PROGRAM PRG_PLAS_15_PrimaryMasterListCtrl
VAR

	bEnablePackMasterListCameraSystem 	: BOOL;

	tofPrimaryMasterListCameraOFFDelay 		: TOF;

	fbShiftMasterListQueue			: FB_PLAS_MasterListShiftQueue;
	fbPrimaryMasterListCamera		: FB_SCANNER_CameraSelect;
	fbPrimaryMasterListEvaluation		: FB_SCANNER_Evaluation;

	fbAddToPrimaryListQueue			: FB_PLAS_MasterListAddToQueue;

	rtrigNewArrived					: R_TRIG;
	bNewCodeIsProccesing			: BOOL;

	tonValidationTimout				: TON;
	bValidationTimeout				: BOOL;
	bValidationTimeoutReset			: BOOL;

	rtPrimaryMasterListCameraDone		:  R_TRIG;
	bPrimaryMasterListCameraDone		:  BOOL;

	fbDebugCNT						: FB_DEBUG_CounterArray;
	aCNTDebug						: ARRAY [1..10] OF UDINT;
	bResetCNT							: BOOL;

END_VAR

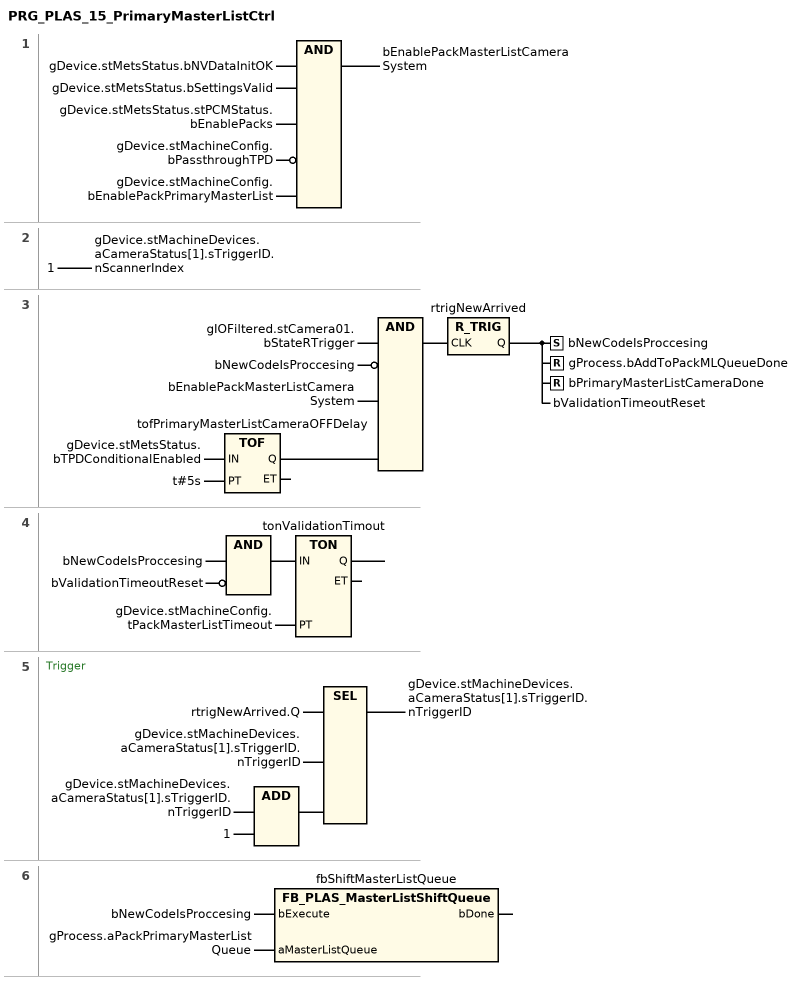
// NETWORK 1
bEnablePackMasterListCameraSystem := gDevice.stMetsStatus.bNVDataInitOK AND gDevice.stMetsStatus.bSettingsValid AND gDevice.stMetsStatus.stPCMStatus.bEnablePacks AND NOT gDevice.stMachineConfig.bPassthroughTPD AND gDevice.stMachineConfig.bEnablePackPrimaryMasterList;

// NETWORK 2
gDevice.stMachineDevices.aCameraStatus[1].sTriggerID.nScannerIndex := 1;

// NETWORK 3
tofPrimaryMasterListCameraOFFDelay(IN := gDevice.stMetsStatus.bTPDConditionalEnabled, PT := t#5s); // TOF
rtrigNewArrived(CLK := gIOFiltered.stCamera01.bStateRTrigger AND NOT bNewCodeIsProccesing AND bEnablePackMasterListCameraSystem AND tofPrimaryMasterListCameraOFFDelay.Q); // R_TRIG
bNewCodeIsProccesing S= rtrigNewArrived.Q;
gProcess.bAddToPackMLQueueDone R= rtrigNewArrived.Q;
bPrimaryMasterListCameraDone R= rtrigNewArrived.Q;
bValidationTimeoutReset := rtrigNewArrived.Q;

// NETWORK 4
tonValidationTimout(IN := bNewCodeIsProccesing AND NOT bValidationTimeoutReset, PT := gDevice.stMachineConfig.tPackMasterListTimeout); // TON

// NETWORK 5
// Trigger
gDevice.stMachineDevices.aCameraStatus[1].sTriggerID.nTriggerID := SEL(rtrigNewArrived.Q, gDevice.stMachineDevices.aCameraStatus[1].sTriggerID.nTriggerID, gDevice.stMachineDevices.aCameraStatus[1].sTriggerID.nTriggerID + 1);

// NETWORK 6
fbShiftMasterListQueue(bExecute := bNewCodeIsProccesing, aMasterListQueue := gProcess.aPackPrimaryMasterListQueue); // FB_PLAS_MasterListShiftQueue

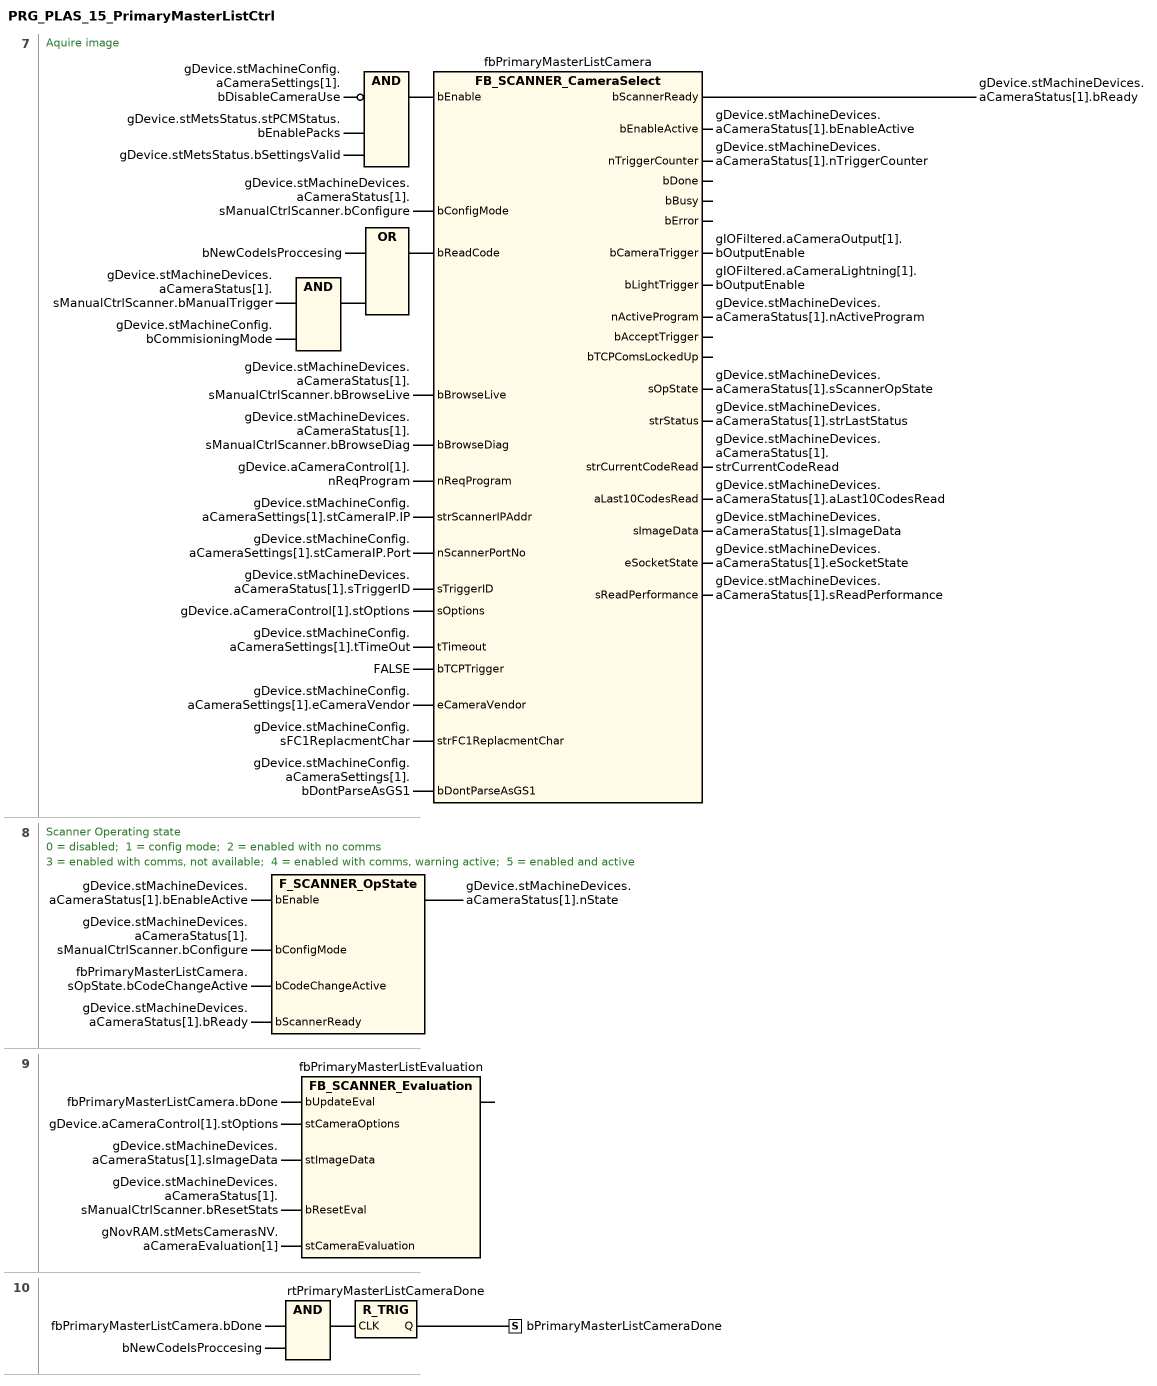
// NETWORK 7
// Aquire image
fbPrimaryMasterListCamera(
    bEnable := NOT gDevice.stMachineConfig.aCameraSettings[1].bDisableCameraUse AND gDevice.stMetsStatus.stPCMStatus.bEnablePacks AND gDevice.stMetsStatus.bSettingsValid,
    bConfigMode := gDevice.stMachineDevices.aCameraStatus[1].sManualCtrlScanner.bConfigure,
    bReadCode := bNewCodeIsProccesing OR gDevice.stMachineDevices.aCameraStatus[1].sManualCtrlScanner.bManualTrigger AND gDevice.stMachineConfig.bCommisioningMode,
    bBrowseLive := gDevice.stMachineDevices.aCameraStatus[1].sManualCtrlScanner.bBrowseLive,
    bBrowseDiag := gDevice.stMachineDevices.aCameraStatus[1].sManualCtrlScanner.bBrowseDiag,
    nReqProgram := gDevice.aCameraControl[1].nReqProgram,
    strScannerIPAddr := gDevice.stMachineConfig.aCameraSettings[1].stCameraIP.IP,
    nScannerPortNo := gDevice.stMachineConfig.aCameraSettings[1].stCameraIP.Port,
    sTriggerID := gDevice.stMachineDevices.aCameraStatus[1].sTriggerID,
    sOptions := gDevice.aCameraControl[1].stOptions,
    tTimeout := gDevice.stMachineConfig.aCameraSettings[1].tTimeOut,
    bTCPTrigger := FALSE,
    eCameraVendor := gDevice.stMachineConfig.aCameraSettings[1].eCameraVendor,
    strFC1ReplacmentChar := gDevice.stMachineConfig.sFC1ReplacmentChar,
    bDontParseAsGS1 := gDevice.stMachineConfig.aCameraSettings[1].bDontParseAsGS1,
    bEnableActive => gDevice.stMachineDevices.aCameraStatus[1].bEnableActive,
    nTriggerCounter => gDevice.stMachineDevices.aCameraStatus[1].nTriggerCounter,
    bCameraTrigger => gIOFiltered.aCameraOutput[1].bOutputEnable,
    bLightTrigger => gIOFiltered.aCameraLightning[1].bOutputEnable,
    nActiveProgram => gDevice.stMachineDevices.aCameraStatus[1].nActiveProgram,
    sOpState => gDevice.stMachineDevices.aCameraStatus[1].sScannerOpState,
    strStatus => gDevice.stMachineDevices.aCameraStatus[1].strLastStatus,
    strCurrentCodeRead => gDevice.stMachineDevices.aCameraStatus[1].strCurrentCodeRead,
    aLast10CodesRead => gDevice.stMachineDevices.aCameraStatus[1].aLast10CodesRead,
    sImageData => gDevice.stMachineDevices.aCameraStatus[1].sImageData,
    eSocketState => gDevice.stMachineDevices.aCameraStatus[1].eSocketState,
    sReadPerformance => gDevice.stMachineDevices.aCameraStatus[1].sReadPerformance); // FB_SCANNER_CameraSelect
gDevice.stMachineDevices.aCameraStatus[1].bReady := fbPrimaryMasterListCamera.bScannerReady;

// NETWORK 8
// 					Scanner Operating state
// 0 = disabled;  1 = config mode;  2 = enabled with no comms
// 3 = enabled with comms, not available;  4 = enabled with comms, warning active;  5 = enabled and active
//
gDevice.stMachineDevices.aCameraStatus[1].nState := F_SCANNER_OpState(bEnable := gDevice.stMachineDevices.aCameraStatus[1].bEnableActive, bConfigMode := gDevice.stMachineDevices.aCameraStatus[1].sManualCtrlScanner.bConfigure, bCodeChangeActive := fbPrimaryMasterListCamera.sOpState.bCodeChangeActive, bScannerReady := gDevice.stMachineDevices.aCameraStatus[1].bReady);

// NETWORK 9
fbPrimaryMasterListEvaluation(
    bUpdateEval := fbPrimaryMasterListCamera.bDone,
    stCameraOptions := gDevice.aCameraControl[1].stOptions,
    stImageData := gDevice.stMachineDevices.aCameraStatus[1].sImageData,
    bResetEval := gDevice.stMachineDevices.aCameraStatus[1].sManualCtrlScanner.bResetStats,
    stCameraEvaluation := gNovRAM.stMetsCamerasNV.aCameraEvaluation[1]); // FB_SCANNER_Evaluation

// NETWORK 10
rtPrimaryMasterListCameraDone(CLK := fbPrimaryMasterListCamera.bDone AND bNewCodeIsProccesing); // R_TRIG
bPrimaryMasterListCameraDone S= rtPrimaryMasterListCameraDone.Q;

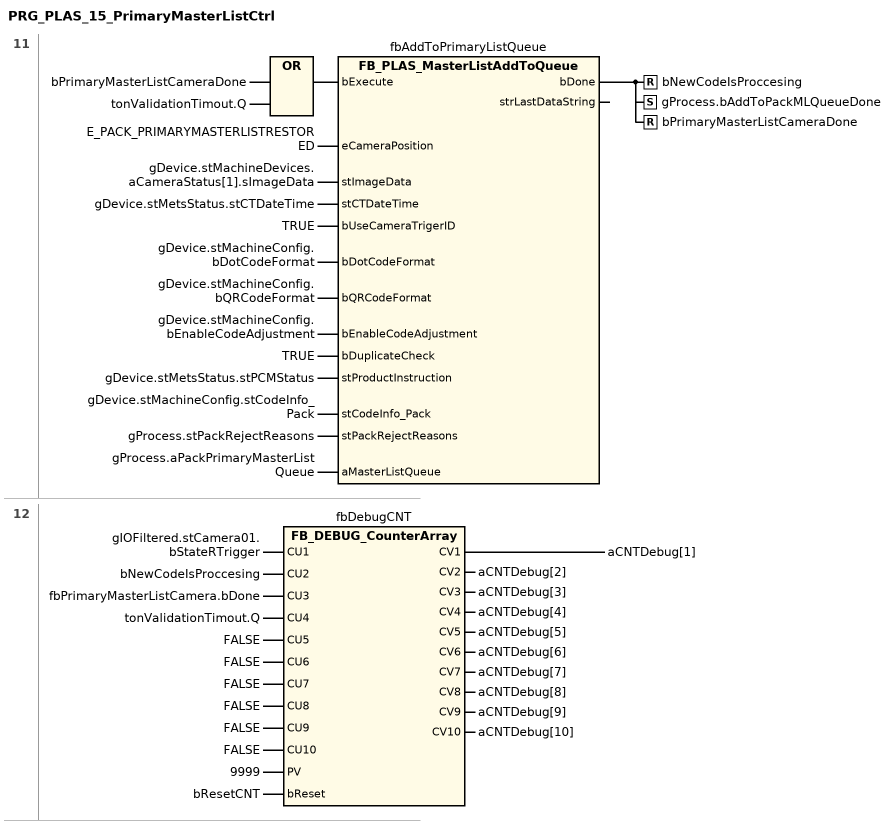
// NETWORK 11
fbAddToPrimaryListQueue(
    bExecute := bPrimaryMasterListCameraDone OR tonValidationTimout.Q,
    eCameraPosition := E_PACK_PRIMARYMASTERLISTRESTORED,
    stImageData := gDevice.stMachineDevices.aCameraStatus[1].sImageData,
    stCTDateTime := gDevice.stMetsStatus.stCTDateTime,
    bUseCameraTrigerID := TRUE,
    bDotCodeFormat := gDevice.stMachineConfig.bDotCodeFormat,
    bQRCodeFormat := gDevice.stMachineConfig.bQRCodeFormat,
    bEnableCodeAdjustment := gDevice.stMachineConfig.bEnableCodeAdjustment,
    bDuplicateCheck := TRUE,
    stProductInstruction := gDevice.stMetsStatus.stPCMStatus,
    stCodeInfo_Pack := gDevice.stMachineConfig.stCodeInfo_Pack,
    stPackRejectReasons := gProcess.stPackRejectReasons,
    aMasterListQueue := gProcess.aPackPrimaryMasterListQueue); // FB_PLAS_MasterListAddToQueue
bNewCodeIsProccesing R= fbAddToPrimaryListQueue.bDone;
gProcess.bAddToPackMLQueueDone S= fbAddToPrimaryListQueue.bDone;
bPrimaryMasterListCameraDone R= fbAddToPrimaryListQueue.bDone;

// NETWORK 12
fbDebugCNT(
    CU1 := gIOFiltered.stCamera01.bStateRTrigger,
    CU2 := bNewCodeIsProccesing,
    CU3 := fbPrimaryMasterListCamera.bDone,
    CU4 := tonValidationTimout.Q,
    CU5 := FALSE,
    CU6 := FALSE,
    CU7 := FALSE,
    CU8 := FALSE,
    CU9 := FALSE,
    CU10 := FALSE,
    PV := 9999,
    bReset := bResetCNT,
    CV2 => aCNTDebug[2],
    CV3 => aCNTDebug[3],
    CV4 => aCNTDebug[4],
    CV5 => aCNTDebug[5],
    CV6 => aCNTDebug[6],
    CV7 => aCNTDebug[7],
    CV8 => aCNTDebug[8],
    CV9 => aCNTDebug[9],
    CV10 => aCNTDebug[10]); // FB_DEBUG_CounterArray
aCNTDebug[1] := fbDebugCNT.CV1;

END_PROGRAM

(* stored: Version 1.1.0.1
   POU PRG_PLAS_15_PrimaryMasterListCtrl: Id {371ee7c4-a150-4819-b714-35d6d285c50b}, SpecialFunc None *)
